KUKA KRL program: wkz3_off_st600.src, wkz3_off_st600.dat

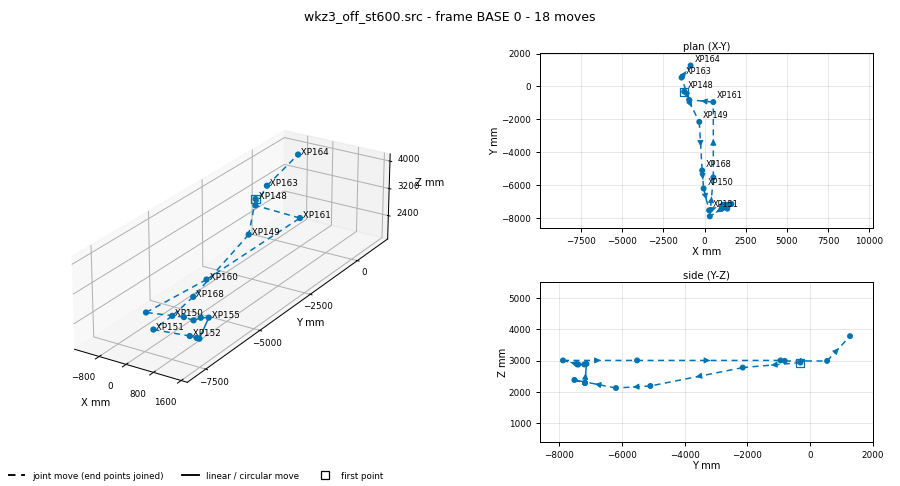
[picture p0: tool path of wkz3_off_st600.src in frame BASE 0, 18 of 19 moves have a stored position in this frame; points joined in program order, loops and branches not executed]
--- wkz3_off_st600.src ---
&ACCESS RVO1
&REL 133
&COMMENT Pega Gripper ACTROS Geobox
&PARAM DISKPATH = KRC:\R1\Program
DEF wkz3_off_st600( )
;FOLD INI
  ;FOLD BASISTECH INI
    GLOBAL INTERRUPT DECL 3 WHEN $STOPMESS==TRUE DO IR_STOPM ( )
    INTERRUPT ON 3
    BAS (#INITMOV,0 )
  ;ENDFOLD (BASISTECH INI)
;FOLD GRIPPERTECH INI
USER_GRP(0,DUMMY,DUMMY,GDEFAULT)
;ENDFOLD (GRIPPERTECH INI)
  ;FOLD USER INI
    ;Make your modifications here

  ;ENDFOLD (USER INI)
;ENDFOLD (INI)

; Caracterização dos meios de produção:
; Versão Atual:
; 12/07/2013 12:00 Name: P13.050-R3 CHANGES: Pega Gripper na Geo
; MGS, MGSB,LTA, LTB e STB

chk_w8_wechs_ok ( )       ; CHECK TOOLCHANGER

;FOLD PTP P148 CONT Vel=100 % PDAT114 Tool[8]:Tool Changer Base[0];%{PE}%R 8.2.20,%MKUKATPBASIS,%CMOVE,%VPTP,%P 1:PTP, 2:P148, 3:C_DIS, 5:100, 7:PDAT114
$BWDSTART=FALSE
PDAT_ACT=PPDAT114
FDAT_ACT=FP148
BAS(#PTP_PARAMS,100)
PTP XP148 C_DIS
;ENDFOLD
;FOLD PTP P149 CONT Vel=100 % PDAT115 Tool[8]:Tool Changer Base[0];%{PE}%R 8.2.20,%MKUKATPBASIS,%CMOVE,%VPTP,%P 1:PTP, 2:P149, 3:C_DIS, 5:100, 7:PDAT115
$BWDSTART=FALSE
PDAT_ACT=PPDAT115
FDAT_ACT=FP149
BAS(#PTP_PARAMS,100)
PTP XP149 C_DIS
;ENDFOLD
;FOLD PTP P168 CONT Vel=100 % PDAT129 Tool[8]:Tool Changer Base[0];%{PE}%R 8.2.20,%MKUKATPBASIS,%CMOVE,%VPTP,%P 1:PTP, 2:P168, 3:C_DIS, 5:100, 7:PDAT129
$BWDSTART=FALSE
PDAT_ACT=PPDAT129
FDAT_ACT=FP168
BAS(#PTP_PARAMS,100)
PTP XP168 C_DIS
;ENDFOLD

;FOLD OUT 3337 'R3 retira garra Geo' State=TRUE ;%{PE}%R 8.2.20,%MKUKATPBASIS,%COUT,%VOUTX,%P 2:3337, 3:R3 retira garra Geo, 5:TRUE, 6:
$OUT[3337]=TRUE
;ENDFOLD
;FOLD WAIT FOR ( IN 3337 'Aguarda Lib. entrar Geo' );%{PE}%R 8.2.20,%MKUKATPBASIS,%CEXT_WAIT_FOR,%VEXT_WAIT_FOR,%P 2:, 4:, 5:$IN, 6:3337, 7:Aguarda Lib. entrar Geo, 9:
WAIT FOR  ( $IN[3337] )
;ENDFOLD
;FOLD OUT 3337 'R3 retira garra Geo' State=FALSE ;%{PE}%R 8.2.20,%MKUKATPBASIS,%COUT,%VOUTX,%P 2:3337, 3:R3 retira garra Geo, 5:FALSE, 6:
$OUT[3337]=FALSE
;ENDFOLD
;FOLD OUT 3338 'R3 solda geometria Ok' State=FALSE ;%{PE}%R 8.2.20,%MKUKATPBASIS,%COUT,%VOUTX,%P 2:3338, 3:R3 solda geometria Ok, 5:FALSE, 6:
$OUT[3338]=FALSE
;ENDFOLD
;FOLD OUT 3348 'Fora area GEOBOX' State=FALSE ;%{PE}%R 8.2.20,%MKUKATPBASIS,%COUT,%VOUTX,%P 2:3348, 3:Fora area GEOBOX, 5:FALSE, 6:
$OUT[3348]=FALSE
;ENDFOLD

;FOLD Collision.Monitoring_1_On ;%{PE}%MKUKATPUSER
COLLSTOP( 1, 1 ) ;Interrupt-Controlled
;ENDFOLD

;FOLD PTP P150 CONT Vel=100 % PDAT116 Tool[8]:Tool Changer Base[0];%{PE}%R 8.2.20,%MKUKATPBASIS,%CMOVE,%VPTP,%P 1:PTP, 2:P150, 3:C_DIS, 5:100, 7:PDAT116
$BWDSTART=FALSE
PDAT_ACT=PPDAT116
FDAT_ACT=FP150
BAS(#PTP_PARAMS,100)
PTP XP150 C_DIS
;ENDFOLD
;FOLD PTP P151 CONT Vel=100 % PDAT117 Tool[8]:Tool Changer Base[0];%{PE}%R 8.2.20,%MKUKATPBASIS,%CMOVE,%VPTP,%P 1:PTP, 2:P151, 3:C_DIS, 5:100, 7:PDAT117
$BWDSTART=FALSE
PDAT_ACT=PPDAT117
FDAT_ACT=FP151
BAS(#PTP_PARAMS,100)
PTP XP151 C_DIS
;ENDFOLD
;FOLD PTP P152 CONT Vel=100 % PDAT118 Tool[8]:Tool Changer Base[0];%{PE}%R 8.2.20,%MKUKATPBASIS,%CMOVE,%VPTP,%P 1:PTP, 2:P152, 3:C_DIS, 5:100, 7:PDAT118
$BWDSTART=FALSE
PDAT_ACT=PPDAT118
FDAT_ACT=FP152
BAS(#PTP_PARAMS,100)
PTP XP152 C_DIS
;ENDFOLD

;FOLD LIN P153 Vel=0.25 m/s CPDAT46 Tool[8]:Tool Changer Base[0];%{PE}%R 8.2.20,%MKUKATPBASIS,%CMOVE,%VLIN,%P 1:LIN, 2:P153, 3:, 5:0.25, 7:CPDAT46
$BWDSTART=FALSE
LDAT_ACT=LCPDAT46
FDAT_ACT=FP153
BAS(#CP_PARAMS,0.25)
LIN XP153
;ENDFOLD

;FOLD OUT 224 'Bloquear MPS' State=FALSE ;%{PE}%R 8.2.20,%MKUKATPBASIS,%COUT,%VOUTX,%P 2:224, 3:Bloquear MPS, 5:FALSE, 6:
$OUT[224]=FALSE
;ENDFOLD
;FOLD OUT 223 'Desbloquear MPS' State=TRUE ;%{PE}%R 8.2.20,%MKUKATPBASIS,%COUT,%VOUTX,%P 2:223, 3:Desbloquear MPS, 5:TRUE, 6:
$OUT[223]=TRUE
;ENDFOLD
;FOLD WAIT FOR ( IN 217 'MPS Destravado' );%{PE}%R 8.2.20,%MKUKATPBASIS,%CEXT_WAIT_FOR,%VEXT_WAIT_FOR,%P 2:, 4:, 5:$IN, 6:217, 7:MPS Destravado, 9:
WAIT FOR  ( $IN[217] )
;ENDFOLD
;FOLD WAIT FOR NOT ( IN 221 'MPS Travado' );%{PE}%R 8.2.20,%MKUKATPBASIS,%CEXT_WAIT_FOR,%VEXT_WAIT_FOR,%P 2:NOT, 4:, 5:$IN, 6:221, 7:MPS Travado, 9:
WAIT FOR  NOT ( $IN[221] )
;ENDFOLD

;FOLD ; PONTO DE PEGA DO GRIPPER;%{PE}%R 5.4.33,%MKUKATPBASIS,%CCOMMENT,%VNORMAL,%P 2:PONTO DE PEGA DO GRIPPER
;ENDFOLD
;FOLD LIN P154 Vel=0.1 m/s CPDAT47 Tool[8]:Tool Changer Base[0];%{PE}%R 8.2.20,%MKUKATPBASIS,%CMOVE,%VLIN,%P 1:LIN, 2:P154, 3:, 5:0.1, 7:CPDAT47
$BWDSTART=FALSE
LDAT_ACT=LCPDAT47
FDAT_ACT=FP154
BAS(#CP_PARAMS,0.1)
LIN XP154
;ENDFOLD

;FOLD WAIT Time=0.5 sec;%{PE}%R 8.2.20,%MKUKATPBASIS,%CWAIT,%VWAIT,%P 3:0.5
WAIT SEC 0.5
;ENDFOLD
;FOLD WAIT FOR ( IN 219 'Posicao p/ Acoplamento OK' );%{PE}%R 8.2.20,%MKUKATPBASIS,%CEXT_WAIT_FOR,%VEXT_WAIT_FOR,%P 2:, 4:, 5:$IN, 6:219, 7:Posicao p/ Acoplamento OK, 9:
WAIT FOR  ( $IN[219] )
;ENDFOLD
;FOLD OUT 223 'Desbloquear MPS' State=FALSE ;%{PE}%R 8.2.20,%MKUKATPBASIS,%COUT,%VOUTX,%P 2:223, 3:Desbloquear MPS, 5:FALSE, 6:
$OUT[223]=FALSE
;ENDFOLD
;FOLD OUT 224 'Bloquear MPS' State=TRUE ;%{PE}%R 8.2.20,%MKUKATPBASIS,%COUT,%VOUTX,%P 2:224, 3:Bloquear MPS, 5:TRUE, 6:
$OUT[224]=TRUE
;ENDFOLD
;FOLD WAIT FOR NOT ( IN 217 'MPS Destravado' );%{PE}%R 8.2.20,%MKUKATPBASIS,%CEXT_WAIT_FOR,%VEXT_WAIT_FOR,%P 2:NOT, 4:, 5:$IN, 6:217, 7:MPS Destravado, 9:
WAIT FOR  NOT ( $IN[217] )
;ENDFOLD
;FOLD WAIT FOR ( IN 221 'MPS Travado' );%{PE}%R 8.2.20,%MKUKATPBASIS,%CEXT_WAIT_FOR,%VEXT_WAIT_FOR,%P 2:, 4:, 5:$IN, 6:221, 7:MPS Travado, 9:
WAIT FOR  ( $IN[221] )
;ENDFOLD
;FOLD IBUS ON SEGMENT_2;%{PE}%R 8.2.20,%MKUKATPBASIS,%CIBUS,%VMAP,%P 2:#ON, 3:2
$IBUS_ON=IBUS_SEGMENT[2]
$IBUS_OFF=0
;ENDFOLD
;FOLD WAIT Time=0.5 sec;%{PE}%R 8.2.20,%MKUKATPBASIS,%CWAIT,%VWAIT,%P 3:0.5
WAIT SEC 0.5
;ENDFOLD

;FOLD OUT 3336 'R3 posição aguardando retirar garra' State=TRUE ;%{PE}%R 8.2.20,%MKUKATPBASIS,%COUT,%VOUTX,%P 2:3336, 3:R3 posição aguardando retirar garra, 5:TRUE, 6:
$OUT[3336]=TRUE
;ENDFOLD
;FOLD WAIT FOR ( IN 3335 'Aguarda Lib. entrar Geo' );%{PE}%R 8.2.20,%MKUKATPBASIS,%CEXT_WAIT_FOR,%VEXT_WAIT_FOR,%P 2:, 4:, 5:$IN, 6:3335, 7:Aguarda Lib. entrar Geo, 9:
WAIT FOR  ( $IN[3335] )
;ENDFOLD
;FOLD OUT 3336 'R3 posição aguardando retirar garra' State=FALSE ;%{PE}%R 8.2.20,%MKUKATPBASIS,%COUT,%VOUTX,%P 2:3336, 3:R3 posição aguardando retirar garra, 5:FALSE, 6:
$OUT[3336]=FALSE
;ENDFOLD

;FOLD SET Z1.1/2 GRP ACTROS State=OPN GDAT11;%{PE}%R 8.2.1,%MKUKATPGRP,%CGRP,%VGRP,%P 2:1, 4:1, 5:#NO, 6:GDAT11, 8:0, 10:0
H50(GRP,1,1,GGDAT11)
;ENDFOLD
;FOLD SET Z2 GRP ACTROS State=OPN GDAT12;%{PE}%R 8.2.1,%MKUKATPGRP,%CGRP,%VGRP,%P 2:2, 4:1, 5:#NO, 6:GDAT12, 8:0, 10:0
H50(GRP,2,1,GGDAT12)
;ENDFOLD
;FOLD SET Z3 GRP ACTROS State=OPN GDAT13;%{PE}%R 8.2.1,%MKUKATPGRP,%CGRP,%VGRP,%P 2:3, 4:1, 5:#NO, 6:GDAT13, 8:0, 10:0
H50(GRP,3,1,GGDAT13)
;ENDFOLD
;FOLD SET Z4.1/2/3/4/5/6/7 ACTROS State=OPN GDAT2;%{PE}%R 8.2.1,%MKUKATPGRP,%CGRP,%VGRP,%P 2:4, 4:1, 5:#NO, 6:GDAT2, 8:0, 10:0
H50(GRP,4,1,GGDAT2)
;ENDFOLD
;FOLD SET Z5 GRP ACTROS State=OPN GDAT14;%{PE}%R 8.2.1,%MKUKATPGRP,%CGRP,%VGRP,%P 2:5, 4:1, 5:#NO, 6:GDAT14, 8:0, 10:0
H50(GRP,5,1,GGDAT14)
;ENDFOLD
    chk_w3_grp1_opn()
    chk_w3_grp2_opn()
    chk_w3_grp3_opn()
    chk_w3_grp4_opn()
    chk_w3_grp5_opn()

;FOLD LIN P155 Vel=0.1 m/s CPDAT48 Tool[3]:Gripper Lateral E.Actros Base[0];%{PE}%R 8.2.20,%MKUKATPBASIS,%CMOVE,%VLIN,%P 1:LIN, 2:P155, 3:, 5:0.1, 7:CPDAT48
$BWDSTART=FALSE
LDAT_ACT=LCPDAT48
FDAT_ACT=FP155
BAS(#CP_PARAMS,0.1)
LIN XP155
;ENDFOLD

;FOLD WAIT FOR ( IN 219 'Posicao p/ Acoplamento OK' ) CONT;%{PE}%R 8.2.20,%MKUKATPBASIS,%CEXT_WAIT_FOR,%VEXT_WAIT_FOR,%P 2:, 4:, 5:$IN, 6:219, 7:Posicao p/ Acoplamento OK, 9:CONTINUE
CONTINUE
WAIT FOR  ( $IN[219] )
;ENDFOLD

;FOLD LIN P156 Vel=0.1 m/s CPDAT49 Tool[3]:Gripper Lateral E.Actros Base[0];%{PE}%R 8.2.20,%MKUKATPBASIS,%CMOVE,%VLIN,%P 1:LIN, 2:P156, 3:, 5:0.1, 7:CPDAT49
$BWDSTART=FALSE
LDAT_ACT=LCPDAT49
FDAT_ACT=FP156
BAS(#CP_PARAMS,0.1)
LIN XP156
;ENDFOLD
;FOLD LIN P157 Vel=0.1 m/s CPDAT50 Tool[3]:Gripper Lateral E.Actros Base[0];%{PE}%R 8.2.20,%MKUKATPBASIS,%CMOVE,%VLIN,%P 1:LIN, 2:P157, 3:, 5:0.1, 7:CPDAT50
$BWDSTART=FALSE
LDAT_ACT=LCPDAT50
FDAT_ACT=FP157
BAS(#CP_PARAMS,0.1)
LIN XP157
;ENDFOLD

;FOLD PTP P158 Vel=100 % PDAT119 Tool[3]:Gripper Lateral E.Actros Base[0];%{PE}%R 8.2.20,%MKUKATPBASIS,%CMOVE,%VPTP,%P 1:PTP, 2:P158, 3:, 5:100, 7:PDAT119
$BWDSTART=FALSE
PDAT_ACT=PPDAT119
FDAT_ACT=FP158
BAS(#PTP_PARAMS,100)
PTP XP158
;ENDFOLD
;FOLD PTP P159 CONT Vel=100 % PDAT120 Tool[8]:Tool Changer Base[0];%{PE}%R 8.2.20,%MKUKATPBASIS,%CMOVE,%VPTP,%P 1:PTP, 2:P159, 3:C_DIS, 5:100, 7:PDAT120
$BWDSTART=FALSE
PDAT_ACT=PPDAT120
FDAT_ACT=FP159
BAS(#PTP_PARAMS,100)
PTP XP159 C_DIS
;ENDFOLD
;FOLD PTP P160 CONT Vel=100 % PDAT121 Tool[8]:Tool Changer Base[0];%{PE}%R 8.2.20,%MKUKATPBASIS,%CMOVE,%VPTP,%P 1:PTP, 2:P160, 3:C_DIS, 5:100, 7:PDAT121
$BWDSTART=FALSE
PDAT_ACT=PPDAT121
FDAT_ACT=FP160
BAS(#PTP_PARAMS,100)
PTP XP160 C_DIS
;ENDFOLD

;FOLD Collision.Monitoring_1_Off . ;%{PE}%MKUKATPUSER
COLLSTOP( 1, 2+0 )
;ENDFOLD
;FOLD PULSE 3335 'R3 retirou garra da Geo' State=TRUE Time=3 sec;%{PE}%R 8.2.20,%MKUKATPBASIS,%COUT,%VPULSE,%P 2:3335, 3:R3 retirou garra da Geo, 5:TRUE, 6:, 8:3
PULSE($OUT[3335], TRUE,3)
;ENDFOLD
;FOLD OUT 3348 'Fora area GEOBOX' State=TRUE ;%{PE}%R 8.2.20,%MKUKATPBASIS,%COUT,%VOUTX,%P 2:3348, 3:Fora area GEOBOX, 5:TRUE, 6:
$OUT[3348]=TRUE
;ENDFOLD

;FOLD PTP P161 CONT Vel=100 % PDAT122 Tool[8]:Tool Changer Base[0];%{PE}%R 8.2.20,%MKUKATPBASIS,%CMOVE,%VPTP,%P 1:PTP, 2:P161, 3:C_DIS, 5:100, 7:PDAT122
$BWDSTART=FALSE
PDAT_ACT=PPDAT122
FDAT_ACT=FP161
BAS(#PTP_PARAMS,100)
PTP XP161 C_DIS
;ENDFOLD
;FOLD PTP P162 CONT Vel=100 % PDAT123 Tool[8]:Tool Changer Base[0];%{PE}%R 8.2.20,%MKUKATPBASIS,%CMOVE,%VPTP,%P 1:PTP, 2:P162, 3:C_DIS, 5:100, 7:PDAT123
$BWDSTART=FALSE
PDAT_ACT=PPDAT123
FDAT_ACT=FP162
BAS(#PTP_PARAMS,100)
PTP XP162 C_DIS
;ENDFOLD
;FOLD PTP P163 CONT Vel=100 % PDAT124 Tool[8]:Tool Changer Base[0];%{PE}%R 8.2.20,%MKUKATPBASIS,%CMOVE,%VPTP,%P 1:PTP, 2:P163, 3:C_DIS, 5:100, 7:PDAT124
$BWDSTART=FALSE
PDAT_ACT=PPDAT124
FDAT_ACT=FP163
BAS(#PTP_PARAMS,100)
PTP XP163 C_DIS
;ENDFOLD
;FOLD PTP P164 CONT Vel=100 % PDAT125 Tool[8]:Tool Changer Base[0];%{PE}%R 8.2.20,%MKUKATPBASIS,%CMOVE,%VPTP,%P 1:PTP, 2:P164, 3:C_DIS, 5:100, 7:PDAT125
$BWDSTART=FALSE
PDAT_ACT=PPDAT125
FDAT_ACT=FP164
BAS(#PTP_PARAMS,100)
PTP XP164 C_DIS
;ENDFOLD

;FOLD PTP HOME Vel=100 % DEFAULT;%{PE}%R 8.2.20,%MKUKATPBASIS,%CMOVE,%VPTP,%P 1:PTP, 2:HOME, 3:, 5:100, 7:DEFAULT
$BWDSTART=FALSE
PDAT_ACT=PDEFAULT
FDAT_ACT=FHOME
BAS(#PTP_PARAMS,100)
$H_POS=XHOME
PTP XHOME
;ENDFOLD

END

--- wkz3_off_st600.dat ---
&ACCESS RVO1
&REL 133
&COMMENT Pega Gripper ACTROS Geobox
&PARAM DISKPATH = KRC:\R1\Program
DEFDAT  wkz3_off_st600
;FOLD EXTERNAL DECLARATIONS;%{PE}%MKUKATPBASIS,%CEXT,%VCOMMON,%P
;FOLD GRIPPERTECH EXT
EXT  H50 (INT  :IN,INT  :IN,INT  :IN,GRP_TYP  :IN )
;ENDFOLD (GRIPPERTECH EXT)
;FOLD SPOTTECH EXT

;ENDFOLD (SPOTTECH EXT)
;FOLD BASISTECH EXT;%{PE}%MKUKATPBASIS,%CEXT,%VEXT,%P
EXT  BAS (BAS_COMMAND  :IN,REAL  :IN )
DECL INT SUCCESS
;ENDFOLD (BASISTECH EXT)
;FOLD USER EXT;%{E}%MKUKATPUSER,%CEXT,%VEXT,%P
;Make your modifications here

;ENDFOLD (USER EXT)
;ENDFOLD (EXTERNAL DECLARATIONS)


;# ============ START PATH : bh_p13050r3_lta_01 =============
DECL BASIS_SUGG_T LAST_BASIS={POINT1[] "P2                      ",POINT2[] "P2                      ",CP_PARAMS[] "CPDAT0                  ",PTP_PARAMS[] "PDAT2                   ",CONT[] "                        ",CP_VEL[] "2.0                     ",PTP_VEL[] "100                     ",SYNC_PARAMS[] "SYNCDAT                 ",SPL_NAME[] "S0                      "}
DECL GRP_SUGG_T LAST_GRP={NUMBER[] "3                       ",STATE[] "1                       ",PARAMS[] "GDAT10                  "}
DECL GRP_TYP GGDAT2={G_APO #NO,GRP_TIME 0.200000003,CTRL #OFF,DLY 0,DST 1}
DECL GRP_TYP GGDAT7={G_APO #NO,GRP_TIME 0.200000003,CTRL #OFF,DLY 0,DST 1}
DECL GRP_TYP GGDAT8={G_APO #NO,GRP_TIME 0.200000003,CTRL #OFF,DLY 0,DST 1}
DECL GRP_TYP GGDAT9={G_APO #NO,GRP_TIME 0.200000003,CTRL #OFF,DLY 0,DST 1}
DECL GRP_TYP GGDAT10={G_APO #NO,GRP_TIME 0.200000003,CTRL #OFF,DLY 0,DST 1}
DECL PDAT PPDAT114={VEL 100.0,ACC 100.0,APO_DIST 100.0,APO_MODE #CDIS}
DECL E6POS XP148={X -1235.52197,Y -311.552094,Z 2940.38989,A 64.7004318,B 6.25024986,C -123.012497,S 2,T 2,E1 757.330811,E2 0.0,E3 0.0,E4 0.0,E5 0.0,E6 0.0}
DECL FDAT FP148={TOOL_NO 8,BASE_NO 0,IPO_FRAME #BASE,POINT2[] " ",TQ_STATE FALSE}
DECL PDAT PPDAT115={VEL 100.0,ACC 100.0,APO_DIST 100.0,APO_MODE #CDIS}
DECL E6POS XP149={X -319.960388,Y -2147.97095,Z 2782.12695,A 160.690994,B 5.30199194,C -131.380493,S 2,T 3,E1 757.329529,E2 0.0,E3 0.0,E4 0.0,E5 0.0,E6 0.0}
DECL FDAT FP149={TOOL_NO 8,BASE_NO 0,IPO_FRAME #BASE,POINT2[] " ",TQ_STATE FALSE}
DECL PDAT PPDAT116={VEL 100.0,ACC 100.0,APO_DIST 100.0,APO_MODE #CDIS}
DECL E6POS XP150={X -56.6846695,Y -6191.46094,Z 2130.31812,A 149.616196,B 9.14294243,C -165.437805,S 2,T 11,E1 4776.96582,E2 0.0,E3 0.0,E4 0.0,E5 0.0,E6 0.0}
DECL FDAT FP150={TOOL_NO 8,BASE_NO 0,IPO_FRAME #BASE,POINT2[] " ",TQ_STATE FALSE}
DECL PDAT PPDAT117={VEL 100.0,ACC 100.0,APO_DIST 100.0,APO_MODE #CDIS}
DECL E6POS XP151={X 276.6492,Y -7516.78906,Z 2388.448,A -120.443001,B -75.749649,C -113.223,S 2,T 43,E1 6265.49805,E2 0.0,E3 0.0,E4 0.0,E5 0.0,E6 0.0}
DECL FDAT FP151={TOOL_NO 8,BASE_NO 0,IPO_FRAME #BASE,POINT2[] " ",TQ_STATE FALSE}
DECL PDAT PPDAT118={VEL 100.0,ACC 100.0,APO_DIST 100.0,APO_MODE #CDIS}
DECL E6POS XP152={X 1114.12903,Y -7180.79883,Z 2291.79712,A -90.1006699,B -74.75383,C -89.8134232,S 2,T 43,E1 6514.04688,E2 0.0,E3 0.0,E4 0.0,E5 0.0,E6 0.0}
DECL FDAT FP152={TOOL_NO 8,BASE_NO 0,IPO_FRAME #BASE,POINT2[] " ",TQ_STATE FALSE}
DECL LDAT LCPDAT46={VEL 2.0,ACC 100.0,APO_DIST 100.0,APO_FAC 50.0,AXIS_VEL 100.0,AXIS_ACC 100.0,ORI_TYP #VAR,CIRC_TYP #BASE,JERK_FAC 50.0,GEAR_JERK 50.0,EXAX_IGN 0}
DECL E6POS XP153={X 1314.45398,Y -7180.50879,Z 2291.95996,A -90.0988617,B -74.7534714,C -89.8143234,S 2,T 43,E1 6514.04688,E2 0.0,E3 0.0,E4 0.0,E5 0.0,E6 0.0}
DECL FDAT FP153={TOOL_NO 8,BASE_NO 0,IPO_FRAME #BASE,POINT2[] " ",TQ_STATE FALSE}
DECL LDAT LCPDAT47={VEL 2.0,ACC 100.0,APO_DIST 100.0,APO_FAC 50.0,AXIS_VEL 100.0,AXIS_ACC 100.0,ORI_TYP #VAR,CIRC_TYP #BASE,JERK_FAC 50.0,GEAR_JERK 50.0,EXAX_IGN 0}
DECL E6POS XP154={X 1393.776,Y -7182.45215,Z 2294.17993,A -90.4568787,B -74.7933731,C -89.8278732,S 2,T 43,E1 6514.06787,E2 0.0,E3 0.0,E4 0.0,E5 0.0,E6 0.0}
DECL FDAT FP154={TOOL_NO 8,BASE_NO 0,IPO_FRAME #BASE,POINT2[] " ",TQ_STATE FALSE}
DECL LDAT LCPDAT48={VEL 2.0,ACC 100.0,APO_DIST 100.0,APO_FAC 50.0,AXIS_VEL 100.0,AXIS_ACC 100.0,ORI_TYP #VAR,CIRC_TYP #BASE,JERK_FAC 50.0,GEAR_JERK 50.0,EXAX_IGN 0}
DECL E6POS XP155={X 1633.91699,Y -7130.41895,Z 2900.91504,A -90.2907562,B 0.165350899,C -89.9555588,S 2,T 43,E1 6514.06787,E2 0.0,E3 0.0,E4 0.0,E5 0.0,E6 0.0}
DECL FDAT FP155={TOOL_NO 3,BASE_NO 0,IPO_FRAME #BASE,POINT2[] " ",TQ_STATE FALSE}
DECL LDAT LCPDAT49={VEL 2.0,ACC 100.0,APO_DIST 100.0,APO_FAC 50.0,AXIS_VEL 100.0,AXIS_ACC 100.0,ORI_TYP #VAR,CIRC_TYP #BASE,JERK_FAC 50.0,GEAR_JERK 50.0,EXAX_IGN 0}
DECL E6POS XP156={X 1451.40503,Y -7202.2832,Z 2881.42993,A -103.146004,B 0.270674199,C -92.0253677,S 2,T 43,E1 6518.90283,E2 0.0,E3 0.0,E4 0.0,E5 0.0,E6 0.0}
DECL FDAT FP156={TOOL_NO 3,BASE_NO 0,IPO_FRAME #BASE,POINT2[] " ",TQ_STATE FALSE}
DECL LDAT LCPDAT50={VEL 2.0,ACC 100.0,APO_DIST 100.0,APO_FAC 50.0,AXIS_VEL 100.0,AXIS_ACC 100.0,ORI_TYP #VAR,CIRC_TYP #BASE,JERK_FAC 50.0,GEAR_JERK 50.0,EXAX_IGN 0}
DECL E6POS XP157={X 1382.14795,Y -7415.31982,Z 2880.19507,A -103.145699,B 0.270470589,C -92.0255127,S 2,T 43,E1 6518.90381,E2 0.0,E3 0.0,E4 0.0,E5 0.0,E6 0.0}
DECL FDAT FP157={TOOL_NO 3,BASE_NO 0,IPO_FRAME #BASE,POINT2[] " ",TQ_STATE FALSE}
DECL PDAT PPDAT119={VEL 100.0,ACC 100.0,APO_DIST 100.0,APO_MODE #CDIS}
DECL E6POS XP158={X 1090.75195,Y -7392.35596,Z 2883.63696,A -102.683998,B 0.211000696,C -91.7751236,S 2,T 43,E1 6518.45117,E2 0.0,E3 0.0,E4 0.0,E5 0.0,E6 0.0}
DECL FDAT FP158={TOOL_NO 3,BASE_NO 0,IPO_FRAME #BASE,POINT2[] " ",TQ_STATE FALSE}
DECL PDAT PPDAT120={VEL 100.0,ACC 100.0,APO_DIST 100.0,APO_MODE #CDIS}
DECL E6POS XP159={X 319.631195,Y -7881.0791,Z 3009.8689,A -124.744202,B 19.1185398,C -97.557373,S 2,T 43,E1 6518.43408,E2 0.0,E3 0.0,E4 0.0,E5 0.0,E6 0.0}
DECL FDAT FP159={TOOL_NO 3,BASE_NO 0,IPO_FRAME #BASE,POINT2[] " ",TQ_STATE FALSE}
DECL PDAT PPDAT121={VEL 100.0,ACC 100.0,APO_DIST 100.0,APO_MODE #CDIS}
DECL E6POS XP160={X 532.35553,Y -5518.01123,Z 3009.86401,A -115.589699,B 19.1185207,C -97.5576019,S 2,T 43,E1 4223.57422,E2 0.0,E3 0.0,E4 0.0,E5 0.0,E6 0.0}
DECL FDAT FP160={TOOL_NO 3,BASE_NO 0,IPO_FRAME #BASE,POINT2[] " ",TQ_STATE FALSE}
DECL PDAT PPDAT122={VEL 100.0,ACC 100.0,APO_DIST 100.0,APO_MODE #CDIS}
DECL E6POS XP161={X 532.343628,Y -945.208618,Z 3009.83496,A -115.589699,B 19.1207504,C -97.5582199,S 2,T 43,E1 -349.285309,E2 0.0,E3 0.0,E4 0.0,E5 0.0,E6 0.0}
DECL FDAT FP161={TOOL_NO 3,BASE_NO 0,IPO_FRAME #BASE,POINT2[] " ",TQ_STATE FALSE}
DECL PDAT PPDAT123={VEL 100.0,ACC 100.0,APO_DIST 100.0,APO_MODE #CDIS}
DECL E6POS XP162={X -937.901672,Y -808.300781,Z 2994.75293,A 178.472595,B 15.1600704,C -101.426498,S 2,T 42,E1 -263.947693,E2 0.0,E3 0.0,E4 0.0,E5 0.0,E6 0.0}
DECL FDAT FP162={TOOL_NO 3,BASE_NO 0,IPO_FRAME #BASE,POINT2[] " ",TQ_STATE FALSE}
DECL PDAT PPDAT124={VEL 100.0,ACC 100.0,APO_DIST 100.0,APO_MODE #CDIS}
DECL E6POS XP163={X -1397.26794,Y 541.47522,Z 2994.75195,A 118.415001,B 15.1602297,C -101.426498,S 2,T 42,E1 -263.947693,E2 0.0,E3 0.0,E4 0.0,E5 0.0,E6 0.0}
DECL FDAT FP163={TOOL_NO 3,BASE_NO 0,IPO_FRAME #BASE,POINT2[] " ",TQ_STATE FALSE}
DECL PDAT PPDAT125={VEL 100.0,ACC 100.0,APO_DIST 100.0,APO_MODE #CDIS}
DECL E6POS XP164={X -845.78363,Y 1272.24402,Z 3784.375,A 58.77174,B 5.0073328,C -70.2537308,S 2,T 42,E1 -245.157394,E2 0.0,E3 0.0,E4 0.0,E5 0.0,E6 0.0}
DECL FDAT FP164={TOOL_NO 3,BASE_NO 0,IPO_FRAME #BASE,POINT2[] " ",TQ_STATE FALSE}
DECL E6POS XP168={X -144.896393,Y -5093.86377,Z 2195.25806,A 148.520294,B 6.76421309,C -164.663895,S 2,T 3,E1 3783.0061,E2 0.0,E3 0.0,E4 0.0,E5 0.0,E6 0.0}
DECL FDAT FP168={TOOL_NO 8,BASE_NO 0,IPO_FRAME #BASE,POINT2[] " ",TQ_STATE FALSE}
DECL PDAT PPDAT129={VEL 100.0,ACC 100.0,APO_DIST 100.0,APO_MODE #CDIS}
DECL GRP_TYP GGDAT11={G_APO #NO,GRP_TIME 0.200000003,CTRL #OFF,DLY 0,DST 1}
DECL GRP_TYP GGDAT12={G_APO #NO,GRP_TIME 0.200000003,CTRL #OFF,DLY 0,DST 1}
DECL GRP_TYP GGDAT13={G_APO #NO,GRP_TIME 0.200000003,CTRL #OFF,DLY 0,DST 1}
DECL GRP_TYP GGDAT14={G_APO #NO,GRP_TIME 0.200000003,CTRL #OFF,DLY 0,DST 1}
DECL E6POS XP174={X 942.72467,Y -141.161697,Z 823.708984,A 179.818893,B 59.8843002,C -89.9199982,S 2,T 43,E1 5735.10791,E2 0.0,E3 0.0,E4 0.0,E5 0.0,E6 0.0}
DECL FDAT FP174={TOOL_NO 5,BASE_NO 3,IPO_FRAME #BASE,POINT2[] " ",TQ_STATE FALSE}
DECL PDAT PPDAT135={VEL 100.0,ACC 100.0,APO_DIST 100.0}
DECL E6POS XP1={X 1395.23401,Y -7181.59082,Z 2293.5769,A -89.9375763,B -74.8767929,C -90.2787933,S 2,T 43,E1 5735.10791,E2 0.0,E3 0.0,E4 0.0,E5 0.0,E6 0.0}
DECL FDAT FP1={TOOL_NO 8,BASE_NO 0,IPO_FRAME #BASE,POINT2[] " ",TQ_STATE FALSE}
DECL PDAT PPDAT1={VEL 100.0,ACC 100.0,APO_DIST 100.0}
DECL E6POS XP2={X 942.76709,Y -141.160599,Z 823.726685,A 179.816299,B 59.8838081,C -89.9213562,S 2,T 43,E1 5735.10791,E2 0.0,E3 0.0,E4 0.0,E5 0.0,E6 0.0}
DECL FDAT FP2={TOOL_NO 5,BASE_NO 3,IPO_FRAME #BASE,POINT2[] " ",TQ_STATE FALSE}
DECL PDAT PPDAT2={VEL 100.0,ACC 100.0,APO_DIST 100.0}
ENDDAT
